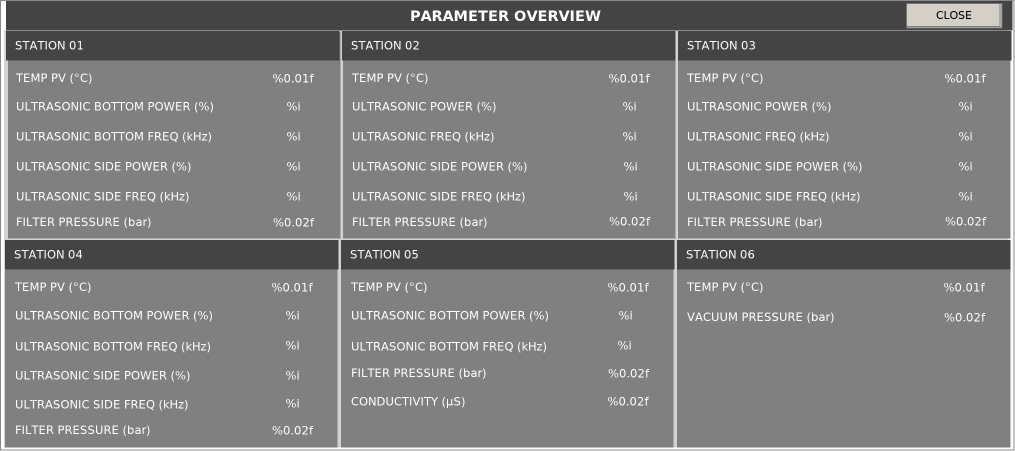
VISUALIZATION Popup_Parameter  // 1015x451
    Rectangle (4,30 1004x417)
    Rectangle (6,1 1006x29)
    Label (407,4 216x24), "PARAMETER OVERVIEW"
    Button (906,3 96x25), "CLOSE"
        OnMouseDown: execute { bParameterPopupPageOn:=0; }
    Rectangle (677,241 333x206)
    Rectangle (677,240 333x29)
    Label (683,242 96x25), "STATION 06"
    Label (684,267 199x40), "TEMP PV (°C)"
    Rectangle (921,264 86x47), "%0.01f", text variable: ARrStnTempPV[6]
    Label (684,296 200x42), "VACUUM PRESSURE (bar)"
    Rectangle (920,297 89x41), "%0.02f", text variable: ARrStnVacuumPV[6]
    Rectangle (8,32 332x206)
    Rectangle (6,31 333x29)
    Label (12,33 96x25), "STATION 01"
    Label (13,58 199x40), "TEMP PV (°C)"
    Rectangle (250,55 86x47), "%0.01f", text variable: ARrStnTempPV[1]
    Label (13,94 235x25), "ULTRASONIC BOTTOM POWER (%)"
    Rectangle (253,93 81x27), "%i", text variable: ARiStnUSBtmAPv[1]
    Label (13,201 163x42), "FILTER PRESSURE (bar)"
    Rectangle (249,202 89x41), "%0.02f", text variable: ARrStnFilterPressurePV[1]
    Label (13,123 240x27), "ULTRASONIC BOTTOM FREQ (kHz)"
    Rectangle (244,117 99x39), "%i", text variable: ARiStnUSBtmAFreqPv[1]
    Label (13,183 240x27), "ULTRASONIC SIDE FREQ (kHz)"
    Label (13,154 235x25), "ULTRASONIC SIDE POWER (%)"
    Rectangle (253,153 81x27), "%i", text variable: ARiStnUSSideAPv[1]
    Rectangle (244,177 99x39), "%i", text variable: ARiStnUSSideAFreqPv[1]
    Rectangle (343,32 332x206)
    Rectangle (342,31 333x29)
    Label (348,33 96x25), "STATION 02"
    Label (349,58 199x40), "TEMP PV (°C)"
    Rectangle (586,55 86x47), "%0.01f", text variable: ARrStnTempPV[2]
    Label (349,94 303x25), "ULTRASONIC POWER (%)"
    Rectangle (589,93 81x27), "%i", text variable: ARiStnUSBtmAPv[2]
    Label (349,201 169x42), "FILTER PRESSURE (bar)"
    Rectangle (585,201 89x41), "%0.02f", text variable: ARrStnFilterPressurePV[2]
    Label (349,123 231x27), "ULTRASONIC FREQ (kHz)"
    Rectangle (580,117 99x39), "%i", text variable: ARiStnUSBtmAFreqPv[2]
    Label (349,154 235x25), "ULTRASONIC SIDE POWER (%)"
    Label (349,183 240x27), "ULTRASONIC SIDE FREQ (kHz)"
    Rectangle (590,153 81x27), "%i", text variable: ARiStnUSSideAPv[2]
    Rectangle (581,177 99x39), "%i", text variable: ARiStnUSSideAFreqPv[2]
    Group (678,31 337x212)
        Rectangle (0,1 332x206)
        Rectangle (0,0 333x29)
        Label (6,2 96x25), "STATION 03"
        Label (6,27 199x40), "TEMP PV (°C)"
        Rectangle (244,24 86x47), "%0.01f", text variable: ARrStnTempPV[3]
        Rectangle (247,62 81x27), "%i", text variable: ARiStnUSBtmAPv[3]
        Label (6,170 165x42), "FILTER PRESSURE (bar)"
        Rectangle (243,170 89x41), "%0.02f", text variable: ARrStnFilterPressurePV[3]
        Label (6,63 173x25), "ULTRASONIC POWER (%)"
        Label (6,92 164x27), "ULTRASONIC FREQ (kHz)"
        Rectangle (238,86 99x39), "%i", text variable: ARiStnUSBtmAFreqPv[3]
        Label (6,123 235x25), "ULTRASONIC SIDE POWER (%)"
        Label (6,152 240x27), "ULTRASONIC SIDE FREQ (kHz)"
        Rectangle (247,122 81x27), "%i", text variable: ARiStnUSSideAPv[1]
        Rectangle (238,146 99x39), "%i", text variable: ARiStnUSSideAFreqPv[1]
    Label (12,332 376x27), "ULTRASONIC FREQ (kHz)"
    Rectangle (5,241 332x206)
    Rectangle (5,240 333x29)
    Label (11,242 96x25), "STATION 04"
    Label (12,267 199x40), "TEMP PV (°C)"
    Rectangle (249,264 86x47), "%0.01f", text variable: ARrStnTempPV[4]
    Label (12,303 232x25), "ULTRASONIC BOTTOM POWER (%)"
    Rectangle (252,302 81x27), "%i", text variable: ARiStnUSBtmAPv[4]
    Label (12,409 170x42), "FILTER PRESSURE (bar)"
    Rectangle (248,410 89x41), "%0.02f", text variable: ARrStnFilterPressurePV[4]
    Rectangle (243,326 99x39), "%i", text variable: ARiStnUSBtmAFreqPv[4]
    Label (12,333 182x27), "ULTRASONIC BOTTOM FREQ (kHz)"
    Label (12,363 201x25), "ULTRASONIC SIDE POWER (%)"
    Rectangle (252,362 81x27), "%i", text variable: ARiStnUSSideAPv[4]
    Rectangle (243,384 99x39), "%i", text variable: ARiStnUSSideAFreqPv[4]
    Label (12,391 210x27), "ULTRASONIC SIDE FREQ (kHz)"
    Group (341,240 341x207)
        Rectangle (0,1 332x206)
        Rectangle (0,0 333x29)
        Label (6,2 96x25), "STATION 05"
        Label (7,27 199x40), "TEMP PV (°C)"
        Rectangle (244,24 86x47), "%0.01f", text variable: ARrStnTempPV[5]
        Label (7,112 165x42), "FILTER PRESSURE (bar)"
        Rectangle (243,113 89x41), "%0.02f", text variable: ARrStnFilterPressurePV[5]
        Label (7,149 173x25), "CONDUCTIVITY (μS)"
        Rectangle (233,152 108x19), "%0.02f", text variable: ARrStnConductivityPV[5]
        Label (7,63 228x25), "ULTRASONIC BOTTOM POWER (%)"
        Rectangle (244,62 81x27), "%i", text variable: ARiStnUSBtmAPv[5]
        Rectangle (234,86 99x39), "%i", text variable: ARiStnUSBtmAFreqPv[5]
        Label (7,93 223x27), "ULTRASONIC BOTTOM FREQ (kHz)"
END_VISUALIZATION

(* stored: Version 1.1.0.1, ProductVersion 3.1.4024.12
   Visu Popup_Parameter: Id {b5b55ea6-9526-49a1-a009-8db01a769e3e} *)
